(* IEC 61131-3 sources: CodesysTest/export/Testing/Actuators/FB_PneumaticVerticalActuator.pou/UpAsserted.prop, 1 file *)

(* ---- Get.pm.st ---- *)
(*#-#-#-#-#-#-#-#-#-#---Declaration---#-#-#-#-#-#-#-#-#-#-#-#-#*)

VAR
END_VAR
(*#-#-#-#-#-#-#-#-#-#---Implementation---#-#-#-#-#-#-#-#-#-#-#-#-#*)

UpAsserted := cylinder.RetractAsserted;
